// TwinCAT 3 PLC project Untitled1
// ProgramVersion: 3.1.4023.0
// libraries:
//   CmpBitmapPool, * (System)
//   Tc2_Standard, * (Beckhoff Automation GmbH)
//   Tc2_System, * (Beckhoff Automation GmbH)
//   Tc3_Module, * (Beckhoff Automation GmbH)
//   VisuDialogs, * (System)
//   VisuSymbols,3.5.10.0,System
// project tree:
//   / GlobalTextList.TcGTLO, PlcTask.TcTTO, Visualization Manager.TcVMO (not stored), VISU_TASK.TcTTO
//   GVLs/ HMI.TcGVL, IO.TcGVL
//   POUs/ MAIN.TcPOU
//   VISUs/ ImagePool.TcIPO (not stored), MainScreen.TcVIS
// real-time tasks:
//   TASK PlcTask: cycle T#10ms, priority 20, ADS port 350
//   TASK VISU_TASK: cycle T#200000us, priority 30, ADS port 351
// I/O:
//   DEVICE Device 1 (EtherCAT), AmsNetId 5.86.83.4.2.1
//     Term 1 (EK1200) [EK1200-5000 EtherCAT Power supply (2A E-Bus)]
//       Term 2 (EL2004) [EL2004 4Ch. Dig. Output 24V, 0.5A]
//       Term 3 (EL3202) [EL3202 2Ch. Ana. Input PT100 (RTD)]
//       Term 4 (EL1008) [EL1008 8Ch. Dig. Input 24V, 3ms]
//       Term 5 (EL1004) [EL1004 4Ch. Dig. Input 24V, 3ms]
//       Term 6 (EL6021) [EL6021 Interface (RS422/485)]
//       Term 7 (EL3314) [EL3314 4Ch. Ana. Input Thermocouple (TC)]
//       Term 8 (EL9011) [EL9011 End Terminal]
// variable links:
//   Untitled1/Untitled1 Instance <-> Device 1 (EtherCAT)/Term 1 (EK1200)/Term 2 (EL2004)
//     PlcTask Outputs/IO.bReactorTu <-> Channel 2/Output
//   Untitled1/Untitled1 Instance <-> Device 1 (EtherCAT)/Term 1 (EK1200)/Term 4 (EL1008)
//     PlcTask Inputs/IO.bReactorHHy <-> Channel 4/Input
//     PlcTask Inputs/IO.bReactorHy <-> Channel 3/Input
//     PlcTask Inputs/IO.bReactorLLy <-> Channel 1/Input
//     PlcTask Inputs/IO.bReactorLy <-> Channel 2/Input
//   Untitled1/Untitled1 Instance <-> Device 1 (EtherCAT)/Term 1 (EK1200)/Term 7 (EL3314)
//     PlcTask Inputs/IO.iInput <-> TC Inputs Channel 1/Value

CONFIGURATION Untitled1
    RESOURCE PLC ON TwinCAT3
        TASK PlcTask(INTERVAL := T#10ms, PRIORITY := 20);
        TASK VISU_TASK(INTERVAL := T#200000us, PRIORITY := 30);
        PROGRAM MAIN WITH PlcTask : MAIN;
        PROGRAM VisuElems_Visu_Prg WITH VISU_TASK : VisuElems.Visu_Prg;
    END_RESOURCE
END_CONFIGURATION

// ---- GVLs/HMI.TcGVL
{attribute 'qualified_only'}
VAR_GLOBAL
	bContactor: BOOL;
	iTemperatureSetpoint: INT; // Temperature controller setpoint
	bTemperatureControlSwitch: BOOL; //Switch for temperature control
	sTemperatureControlState: STRING(35); //Temperature control switch state in str
	iTemperatureDisplayValue: INT; //Displayed temp value in HMI (see MAIN)
	iTemperatureControlPercentage: INT; //Temperature controller output % (0-100)
	
	bLevelControlSwitch: BOOL; //Switch for level control	
	sLevelControlState: STRING(35); //Level control switch state in str
	
	
END_VAR

// ---- GVLs/IO.TcGVL
{attribute 'qualified_only'}
VAR_GLOBAL
	//Test
	{attribute 'OPC.UA.DA' := '1'}
	iInput AT %I* : INT; // Thermocouple test
	bReactorTu AT %Q* : BOOL; // Temperature contactor
	iReactorTy AT %I*: INT; // Reactor temperature
	bReactorHHy AT %I*: BOOL; // Higher high slurry level
	bReactorHy AT %I*: BOOL; // High slurry level
	bReactorLy AT %I*: BOOL; // Low slurry level
	bReactorLLy AT %I*: BOOL; // Lower low slurry level
	bReactorLu AT %Q*: BOOL;  // Reactor outlet valve
	
END_VAR

// ---- POUs/MAIN.TcPOU
PROGRAM MAIN
VAR
END_VAR

//IO.bOutput := HMI.bContactor;
HMI.iTemperatureDisplayValue := IO.iInput/10;
//Temperature Control state
IF HMI.bTemperatureControlSwitch = 1 THEN
	HMI.sTemperatureControlState := 'AUTO';
END_IF
IF HMI.bTemperatureControlSwitch = 0 THEN
	HMI.sTemperatureControlState := 'MAN';
END_IF

END_PROGRAM

// ---- GlobalTextList.TcGTLO
TEXTLIST GlobalTextList
  574 = '%2.0f'
  759 = '%2f'
  655 = '%i'
  23 = '%i *C'
  615 = '%s'
  917 = '&i'
  757 = 'Contactor'
  153 = 'Control'
  154 = 'Label'
  69 = 'Mode'
  351 = 'ON/OFF'
  463 = 'Percentage'
  443 = 'Percentage (%)'
  951 = 'Reactor'
  579 = 'Screen'
  31 = 'Screen1'
  465 = 'Screen2'
  160 = 'Setpoint'
  640 = 'Temperature'
  968 = 'Temperature Control'
END_TEXTLIST

// ---- VISUs/MainScreen.TcVIS
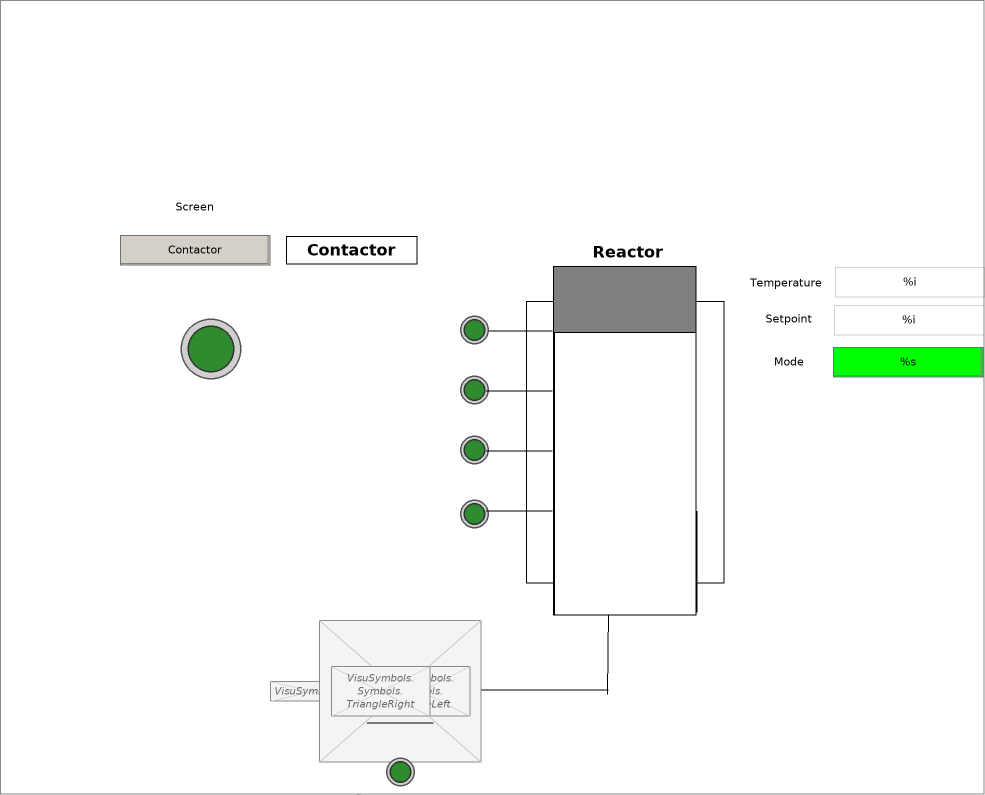
VISUALIZATION MainScreen  // 985x795
    Rectangle (526,301 198x282), colour toggle: HMI.bTemperatureControlSwitch
    RoundedRectangle (553,266 143x345)
    Label (120,192 150x30), "Screen"
    Button (120,235 150x30), "Contactor", colour toggle: HMI.bContactor
        toggle IO.bReactorTu
    Lamp1 (176,314 70x70), variable: IO.bReactorTu, style: Lamp-Lamp1-Green
    Line (552,331) (486,331)
    Lamp1 (458,311 33x38), variable: IO.bReactorHHy, style: Lamp-Lamp1-Green
    Lamp1 (458,371 33x38), variable: IO.bReactorHy, style: Lamp-Lamp1-Green
    Lamp1 (458,431 33x38), variable: IO.bReactorLy, style: Lamp-Lamp1-Green
    Lamp1 (458,495 33x38), variable: IO.bReactorLLy, style: Lamp-Lamp1-Green
    Textfield (834,305 150x30), "%i", text variable: HMI.iTemperatureSetpoint
        OnMouseDown: write the text variable via VisuDialogs.Numpad, min 40, max 120
    Label (715,261 142x44), "Temperature"
    Button (833,347 150x30), "%s", text variable: HMI.sTemperatureControlState, colour toggle: HMI.bTemperatureControlSwitch
        toggle HMI.bTemperatureControlSwitch
    Label (718,340 142x44), "Mode"
    Label (718,297 142x44), "Setpoint"
    Textfield (835,267 150x30), "%i", text variable: HMI.iTemperatureDisplayValue
    Line (608,611) (607,694)
    Line (608,690) (442,690)
    Line (552,391) (486,391)
    Line (552,451) (486,451)
    Line (552,511) (486,511)
    RoundedRectangle (286,236 131x28), "Contactor", invisible if: (NOT IO.bReactorTu) AND (NOT IO.bReactorHHy)
    RoundedRectangle (553,511 144x101), invisible if: (NOT IO.bReactorLLy) OR (IO.bReactorLy)
    Label (553,237 150x30), "Reactor"
    RoundedRectangle (553,452 143x162), invisible if: (NOT IO.bReactorLy) OR (IO.bReactorHy)
    RoundedRectangle (553,392 143x223), invisible if: (NOT IO.bReactorHy) OR (IO.bReactorHHy)
    RoundedRectangle (554,332 142x283), invisible if: (NOT IO.bReactorHHy)
    Image (270,681 83x20), image: VisuSymbols.Symbols.ArrowBoldLeft
    Image (319,620 162x142), invisible if: NOT IO.bReactorLu, image: ImagePool.VALVE
    Image (371,666 99x50), invisible if: IO.bReactorLu, image: VisuSymbols.Symbols.TriangleLeft
    Image (357,794 3x1), image: VisuSymbols.Symbols.TriangleRight
    Image (331,666 99x50), invisible if: IO.bReactorLu, image: VisuSymbols.Symbols.TriangleRight
    Line (433,723) (367,723)
    Lamp1 (384,753 33x38), variable: IO.bReactorLu, style: Lamp-Lamp1-Green
END_VISUALIZATION
